KUKA KRL program: auto_mode.src

&ACCESS RV
DEF auto_mode ( )

END
